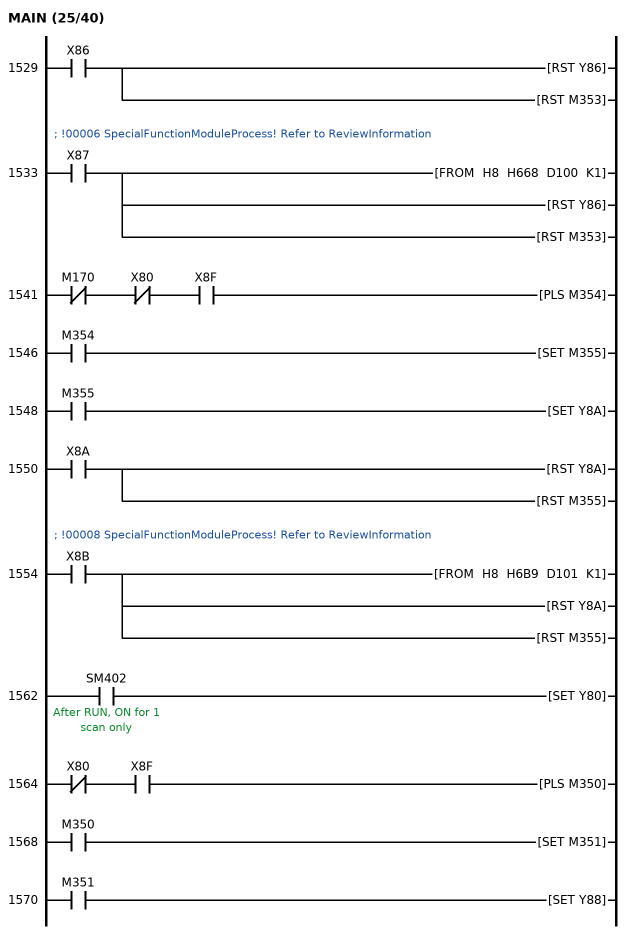
[picture p24: ladder of MAIN, rungs at steps 1529 to 1570]
1529  LD      X86
      RST     Y86
      RST     M353
; !00006 SpecialFunctionModuleProcess! Refer to ReviewInformation
1533  LD      X87
      FROM    H8 H668 D100 K1
      RST     Y86
      RST     M353
1541  LDI     M170
      ANI     X80
      AND     X8F
      PLS     M354
1546  LD      M354
      SET     M355
1548  LD      M355
      SET     Y8A
1550  LD      X8A
      RST     Y8A
      RST     M355
; !00008 SpecialFunctionModuleProcess! Refer to ReviewInformation
1554  LD      X8B
      FROM    H8 H6B9 D101 K1
      RST     Y8A
      RST     M355
1562  LD      SM402  ; After RUN, ON for 1 scan only
      SET     Y80
1564  LDI     X80
      AND     X8F
      PLS     M350
1568  LD      M350
      SET     M351
1570  LD      M351
      SET     Y88
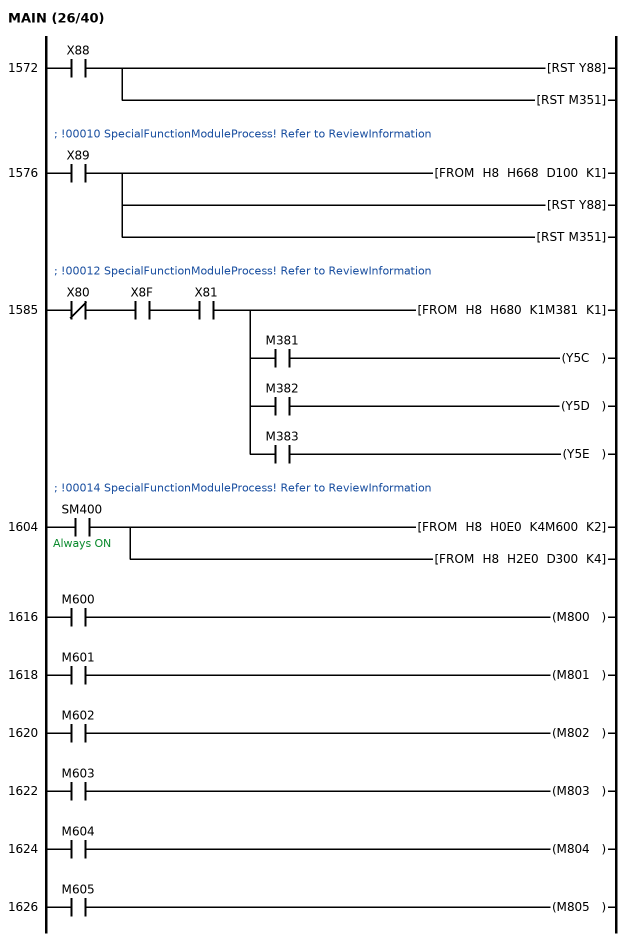
1572  LD      X88
      RST     Y88
      RST     M351
; !00010 SpecialFunctionModuleProcess! Refer to ReviewInformation
1576  LD      X89
      FROM    H8 H668 D100 K1
      RST     Y88
      RST     M351
; !00012 SpecialFunctionModuleProcess! Refer to ReviewInformation
1585  LDI     X80
      AND     X8F
      AND     X81
      FROM    H8 H680 K1M381 K1
      MPS
      AND     M381
      OUT     Y5C
      MRD
      AND     M382
      OUT     Y5D
      MPP
      AND     M383
      OUT     Y5E
; !00014 SpecialFunctionModuleProcess! Refer to ReviewInformation
1604  LD      SM400  ; Always ON
      FROM    H8 H0E0 K4M600 K2
      FROM    H8 H2E0 D300 K4
1616  LD      M600
      OUT     M800
1618  LD      M601
      OUT     M801
1620  LD      M602
      OUT     M802
1622  LD      M603
      OUT     M803
1624  LD      M604
      OUT     M804
1626  LD      M605
      OUT     M805
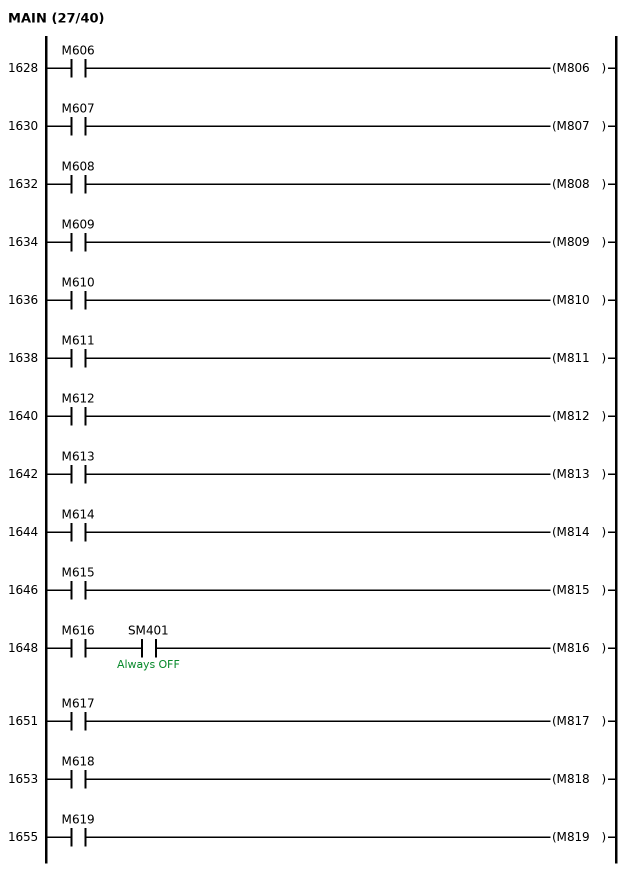
1628  LD      M606
      OUT     M806
1630  LD      M607
      OUT     M807
1632  LD      M608
      OUT     M808
1634  LD      M609
      OUT     M809
1636  LD      M610
      OUT     M810
1638  LD      M611
      OUT     M811
1640  LD      M612
      OUT     M812
1642  LD      M613
      OUT     M813
1644  LD      M614
      OUT     M814
1646  LD      M615
      OUT     M815
1648  LD      M616
      AND     SM401  ; Always OFF
      OUT     M816
1651  LD      M617
      OUT     M817
1653  LD      M618
      OUT     M818
1655  LD      M619
      OUT     M819
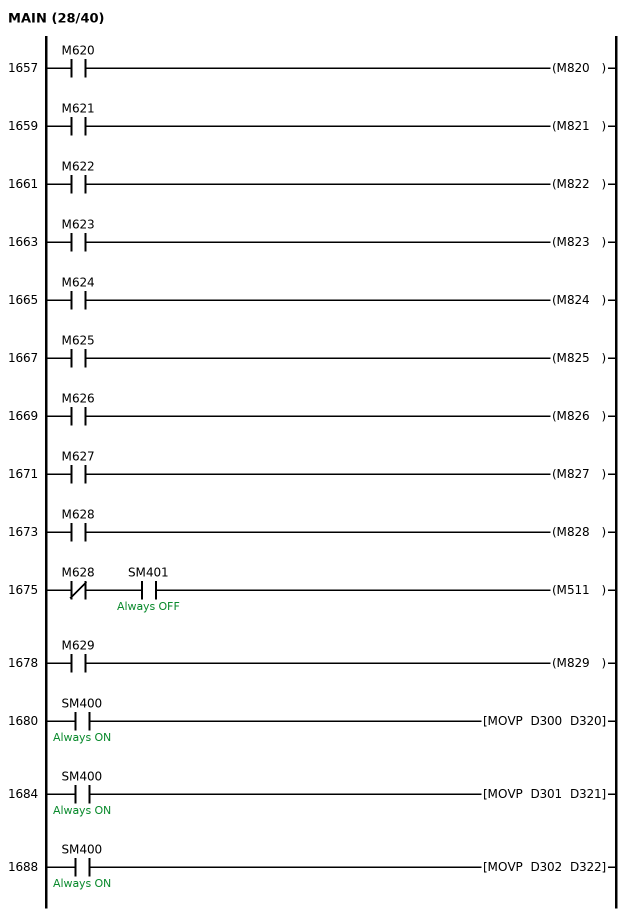
1657  LD      M620
      OUT     M820
1659  LD      M621
      OUT     M821
1661  LD      M622
      OUT     M822
1663  LD      M623
      OUT     M823
1665  LD      M624
      OUT     M824
1667  LD      M625
      OUT     M825
1669  LD      M626
      OUT     M826
1671  LD      M627
      OUT     M827
1673  LD      M628
      OUT     M828
1675  LDI     M628
      AND     SM401  ; Always OFF
      OUT     M511
1678  LD      M629
      OUT     M829
1680  LD      SM400  ; Always ON
      MOVP    D300 D320
1684  LD      SM400  ; Always ON
      MOVP    D301 D321
1688  LD      SM400  ; Always ON
      MOVP    D302 D322
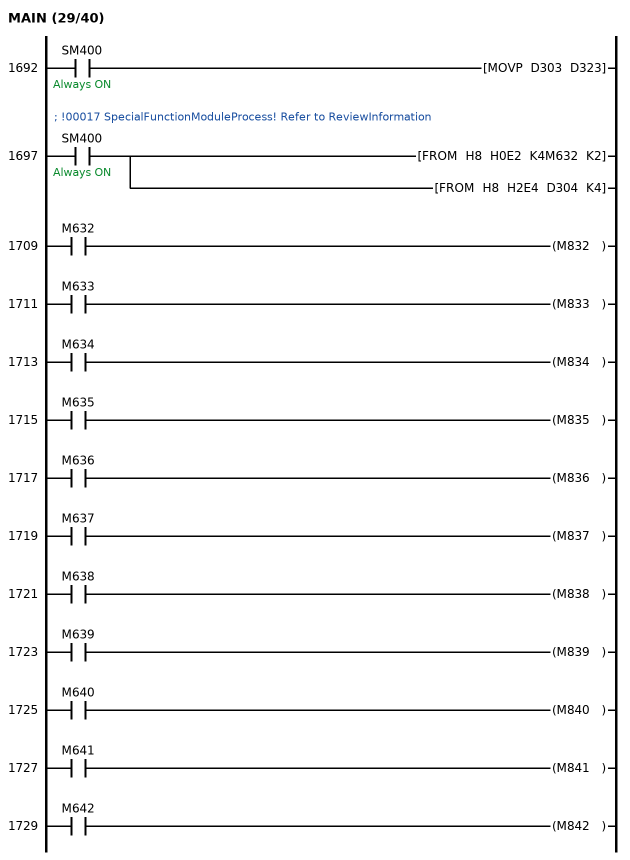
1692  LD      SM400  ; Always ON
      MOVP    D303 D323
; !00017 SpecialFunctionModuleProcess! Refer to ReviewInformation
1697  LD      SM400  ; Always ON
      FROM    H8 H0E2 K4M632 K2
      FROM    H8 H2E4 D304 K4
1709  LD      M632
      OUT     M832
1711  LD      M633
      OUT     M833
1713  LD      M634
      OUT     M834
1715  LD      M635
      OUT     M835
1717  LD      M636
      OUT     M836
1719  LD      M637
      OUT     M837
1721  LD      M638
      OUT     M838
1723  LD      M639
      OUT     M839
1725  LD      M640
      OUT     M840
1727  LD      M641
      OUT     M841
1729  LD      M642
      OUT     M842
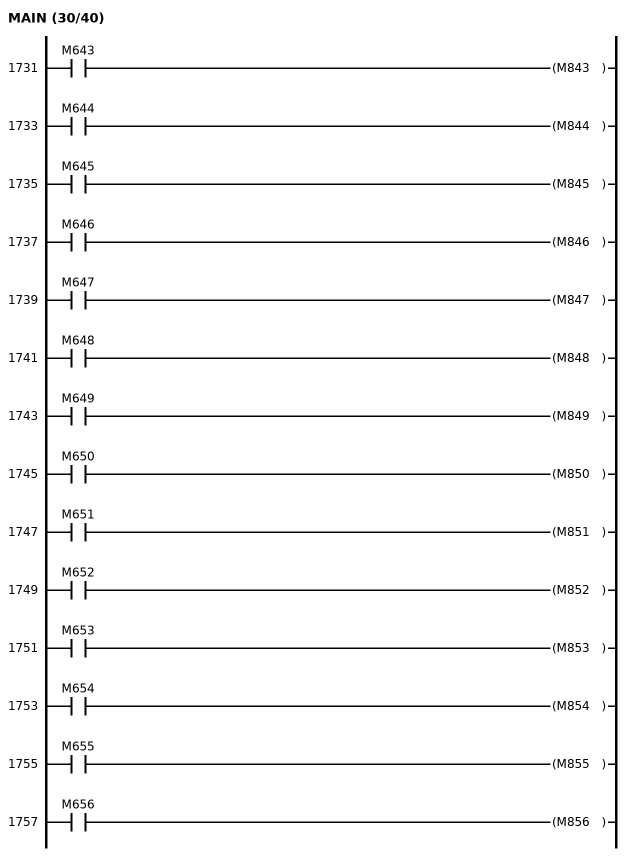
1731  LD      M643
      OUT     M843
1733  LD      M644
      OUT     M844
1735  LD      M645
      OUT     M845
1737  LD      M646
      OUT     M846
1739  LD      M647
      OUT     M847
1741  LD      M648
      OUT     M848
1743  LD      M649
      OUT     M849
1745  LD      M650
      OUT     M850
1747  LD      M651
      OUT     M851
1749  LD      M652
      OUT     M852
1751  LD      M653
      OUT     M853
1753  LD      M654
      OUT     M854
1755  LD      M655
      OUT     M855
1757  LD      M656
      OUT     M856
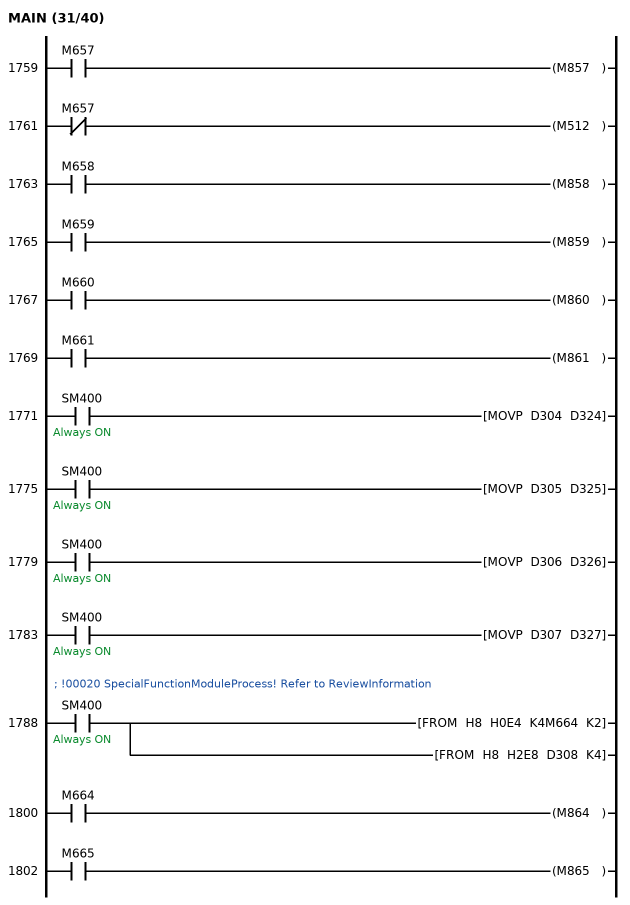
1759  LD      M657
      OUT     M857
1761  LDI     M657
      OUT     M512
1763  LD      M658
      OUT     M858
1765  LD      M659
      OUT     M859
1767  LD      M660
      OUT     M860
1769  LD      M661
      OUT     M861
1771  LD      SM400  ; Always ON
      MOVP    D304 D324
1775  LD      SM400  ; Always ON
      MOVP    D305 D325
1779  LD      SM400  ; Always ON
      MOVP    D306 D326
1783  LD      SM400  ; Always ON
      MOVP    D307 D327
; !00020 SpecialFunctionModuleProcess! Refer to ReviewInformation
1788  LD      SM400  ; Always ON
      FROM    H8 H0E4 K4M664 K2
      FROM    H8 H2E8 D308 K4
1800  LD      M664
      OUT     M864
1802  LD      M665
      OUT     M865
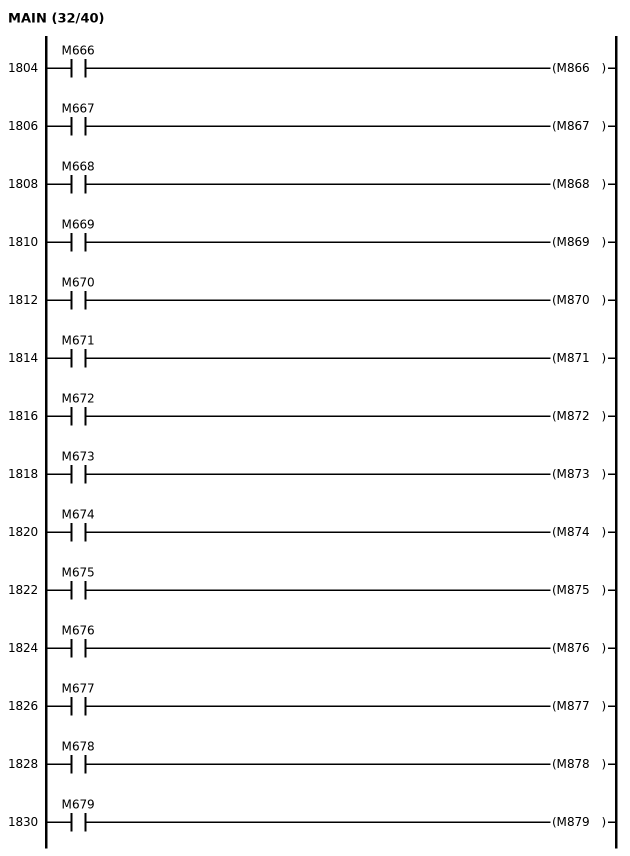
1804  LD      M666
      OUT     M866
1806  LD      M667
      OUT     M867
1808  LD      M668
      OUT     M868
1810  LD      M669
      OUT     M869
1812  LD      M670
      OUT     M870
1814  LD      M671
      OUT     M871
1816  LD      M672
      OUT     M872
1818  LD      M673
      OUT     M873
1820  LD      M674
      OUT     M874
1822  LD      M675
      OUT     M875
1824  LD      M676
      OUT     M876
1826  LD      M677
      OUT     M877
1828  LD      M678
      OUT     M878
1830  LD      M679
      OUT     M879
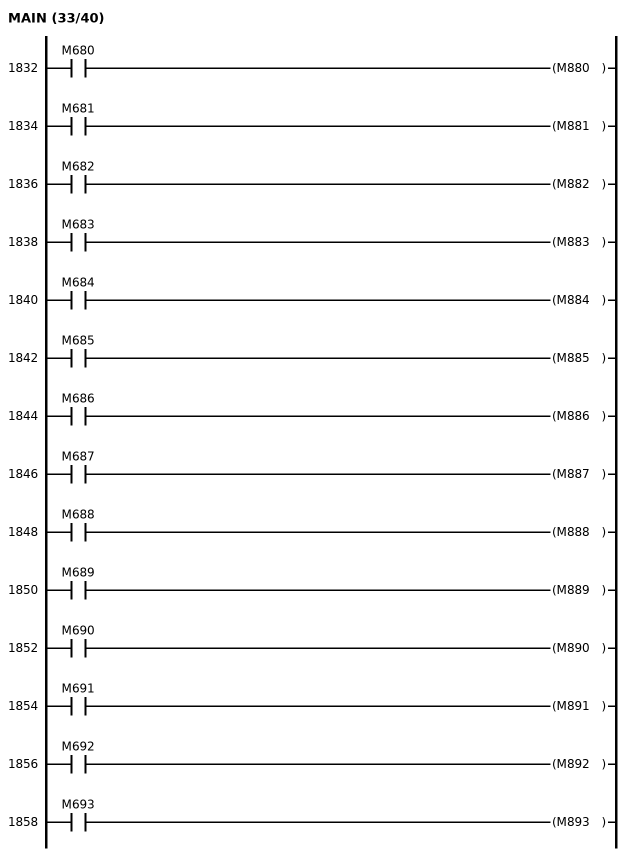
1832  LD      M680
      OUT     M880
1834  LD      M681
      OUT     M881
1836  LD      M682
      OUT     M882
1838  LD      M683
      OUT     M883
1840  LD      M684
      OUT     M884
1842  LD      M685
      OUT     M885
1844  LD      M686
      OUT     M886
1846  LD      M687
      OUT     M887
1848  LD      M688
      OUT     M888
1850  LD      M689
      OUT     M889
1852  LD      M690
      OUT     M890
1854  LD      M691
      OUT     M891
1856  LD      M692
      OUT     M892
1858  LD      M693
      OUT     M893
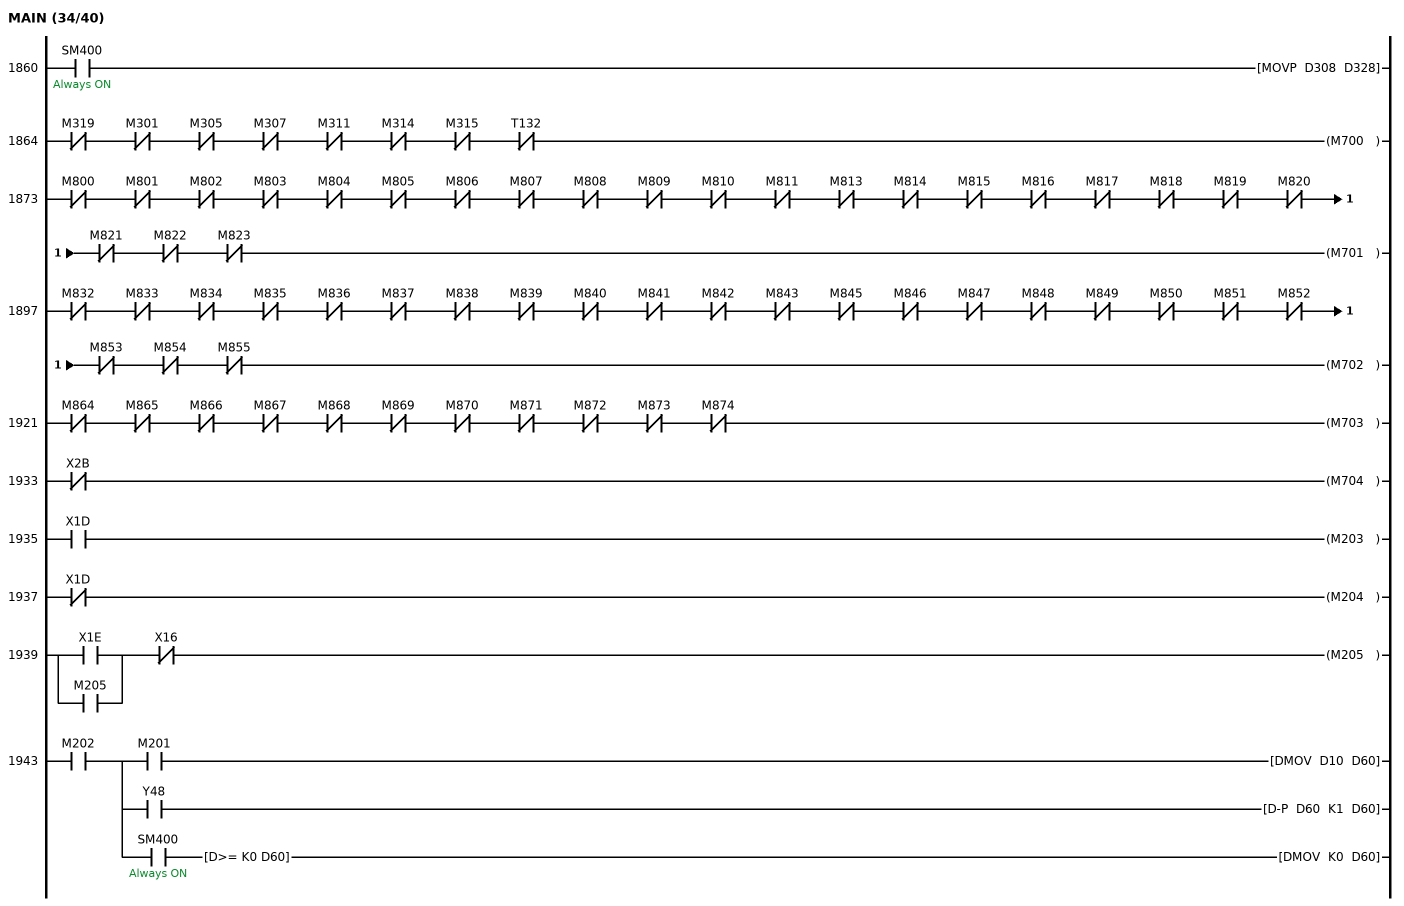
1860  LD      SM400  ; Always ON
      MOVP    D308 D328
1864  LDI     M319
      ANI     M301
      ANI     M305
      ANI     M307
      ANI     M311
      ANI     M314
      ANI     M315
      ANI     T132
      OUT     M700
1873  LDI     M800
      ANI     M801
      ANI     M802
      ANI     M803
      ANI     M804
      ANI     M805
      ANI     M806
      ANI     M807
      ANI     M808
      ANI     M809
      ANI     M810
      ANI     M811
      ANI     M813
      ANI     M814
      ANI     M815
      ANI     M816
      ANI     M817
      ANI     M818
      ANI     M819
      ANI     M820
      ANI     M821
      ANI     M822
      ANI     M823
      OUT     M701
1897  LDI     M832
      ANI     M833
      ANI     M834
      ANI     M835
      ANI     M836
      ANI     M837
      ANI     M838
      ANI     M839
      ANI     M840
      ANI     M841
      ANI     M842
      ANI     M843
      ANI     M845
      ANI     M846
      ANI     M847
      ANI     M848
      ANI     M849
      ANI     M850
      ANI     M851
      ANI     M852
      ANI     M853
      ANI     M854
      ANI     M855
      OUT     M702
1921  LDI     M864
      ANI     M865
      ANI     M866
      ANI     M867
      ANI     M868
      ANI     M869
      ANI     M870
      ANI     M871
      ANI     M872
      ANI     M873
      ANI     M874
      OUT     M703
1933  LDI     X2B
      OUT     M704
1935  LD      X1D
      OUT     M203
1937  LDI     X1D
      OUT     M204
1939  LD      X1E
      OR      M205
      ANI     X16
      OUT     M205
1943  LD      M202
      MPS
      AND     M201
      DMOV    D10 D60
      MRD
      AND     Y48
      D-P     D60 K1 D60
      MPP
      AND     SM400  ; Always ON
      ANDD>=  K0 D60
      DMOV    K0 D60
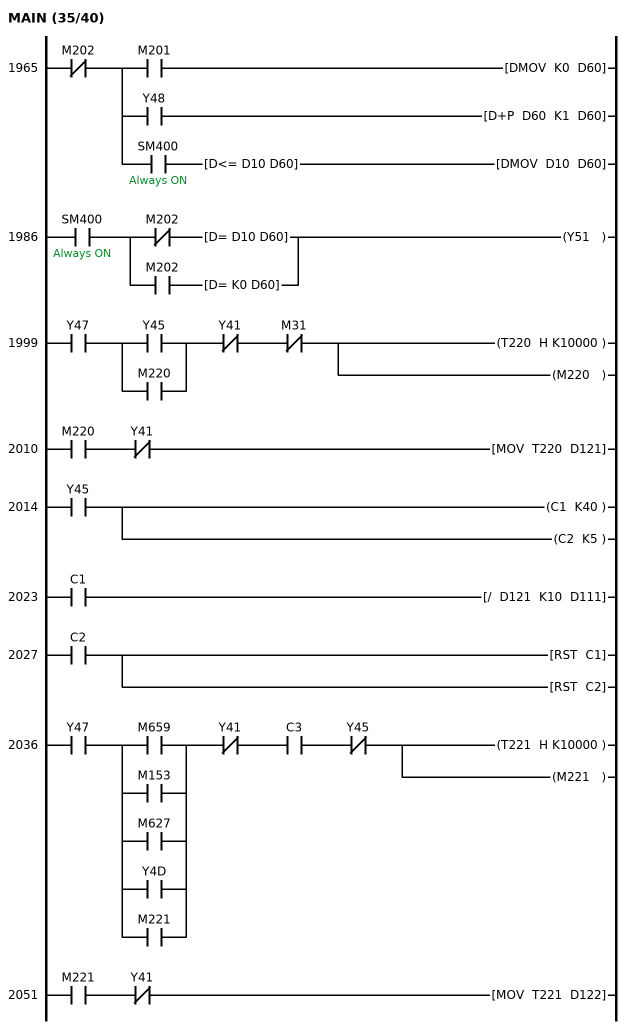
1965  LDI     M202
      MPS
      AND     M201
      DMOV    K0 D60
      MRD
      AND     Y48
      D+P     D60 K1 D60
      MPP
      AND     SM400  ; Always ON
      ANDD<=  D10 D60
      DMOV    D10 D60
1986  LD      SM400  ; Always ON
      LDI     M202
      ANDD=   D10 D60
      LD      M202
      ANDD=   K0 D60
      ORB
      ANB
      OUT     Y51
1999  LD      Y47
      LD      Y45
      OR      M220
      ANB
      ANI     Y41
      ANI     M31
      OUTH    T220 K10000
      OUT     M220
2010  LD      M220
      ANI     Y41
      MOV     T220 D121
2014  LD      Y45
      OUT     C1 K40
      OUT     C2 K5
2023  LD      C1
      /       D121 K10 D111
2027  LD      C2
      RST     C1
      RST     C2
2036  LD      Y47
      LD      M659
      OR      M153
      OR      M627
      OR      Y4D
      OR      M221
      ANB
      ANI     Y41
      AND     C3
      ANI     Y45
      OUTH    T221 K10000
      OUT     M221
2051  LD      M221
      ANI     Y41
      MOV     T221 D122
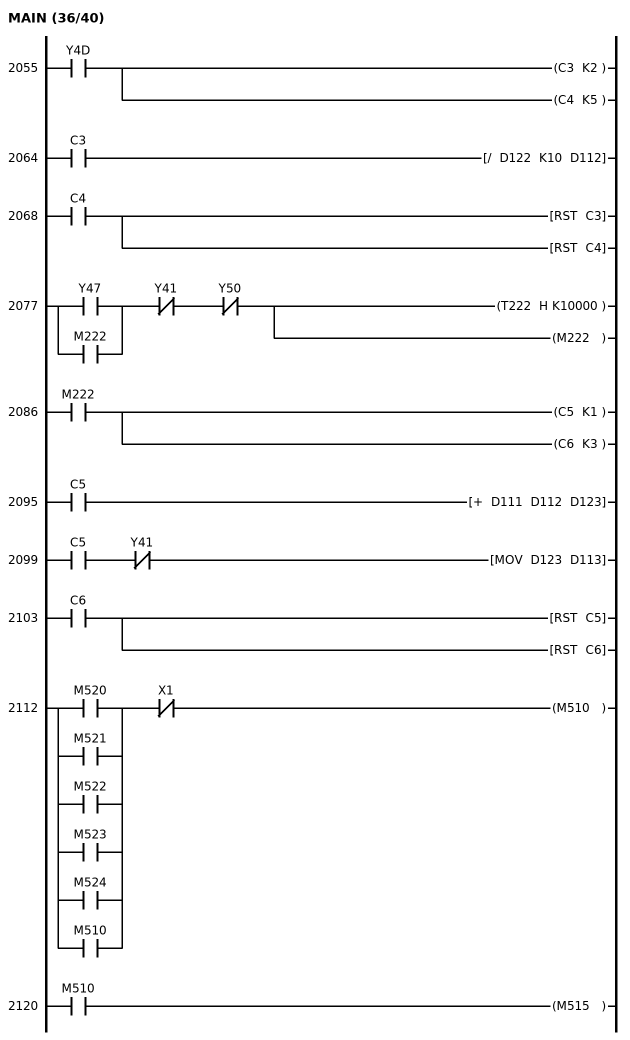
2055  LD      Y4D
      OUT     C3 K2
      OUT     C4 K5
2064  LD      C3
      /       D122 K10 D112
2068  LD      C4
      RST     C3
      RST     C4
2077  LD      Y47
      OR      M222
      ANI     Y41
      ANI     Y50
      OUTH    T222 K10000
      OUT     M222
2086  LD      M222
      OUT     C5 K1
      OUT     C6 K3
2095  LD      C5
      +       D111 D112 D123
2099  LD      C5
      ANI     Y41
      MOV     D123 D113
2103  LD      C6
      RST     C5
      RST     C6
2112  LD      M520
      OR      M521
      OR      M522
      OR      M523
      OR      M524
      OR      M510
      ANI     X1
      OUT     M510
2120  LD      M510
      OUT     M515
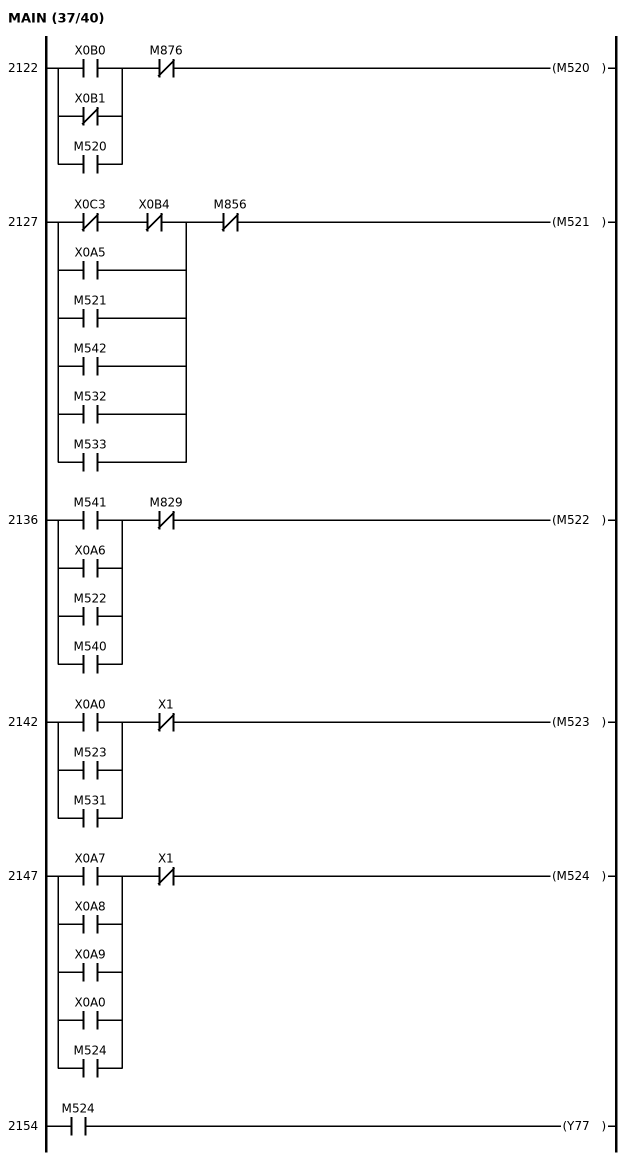
2122  LD      X0B0
      ORI     X0B1
      OR      M520
      ANI     M876
      OUT     M520
2127  LDI     X0C3
      ANI     X0B4
      OR      X0A5
      OR      M521
      OR      M542
      OR      M532
      OR      M533
      ANI     M856
      OUT     M521
2136  LD      M541
      OR      X0A6
      OR      M522
      OR      M540
      ANI     M829
      OUT     M522
2142  LD      X0A0
      OR      M523
      OR      M531
      ANI     X1
      OUT     M523
2147  LD      X0A7
      OR      X0A8
      OR      X0A9
      OR      X0A0
      OR      M524
      ANI     X1
      OUT     M524
2154  LD      M524
      OUT     Y77
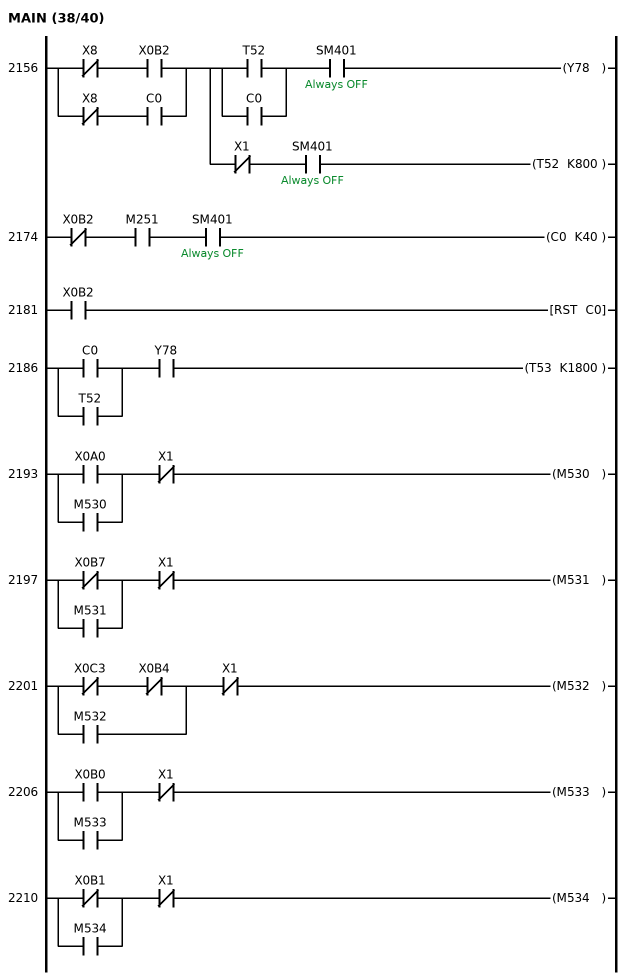
2156  LDI     X8
      AND     X0B2
      LDI     X8
      AND     C0
      ORB
      MPS
      LD      T52
      OR      C0
      ANB
      AND     SM401  ; Always OFF
      OUT     Y78
      MPP
      ANI     X1
      AND     SM401  ; Always OFF
      OUT     T52 K800
2174  LDI     X0B2
      AND     M251
      AND     SM401  ; Always OFF
      OUT     C0 K40
2181  LD      X0B2
      RST     C0
2186  LD      C0
      OR      T52
      AND     Y78
      OUT     T53 K1800
2193  LD      X0A0
      OR      M530
      ANI     X1
      OUT     M530
2197  LDI     X0B7
      OR      M531
      ANI     X1
      OUT     M531
2201  LDI     X0C3
      ANI     X0B4
      OR      M532
      ANI     X1
      OUT     M532
2206  LD      X0B0
      OR      M533
      ANI     X1
      OUT     M533
2210  LDI     X0B1
      OR      M534
      ANI     X1
      OUT     M534
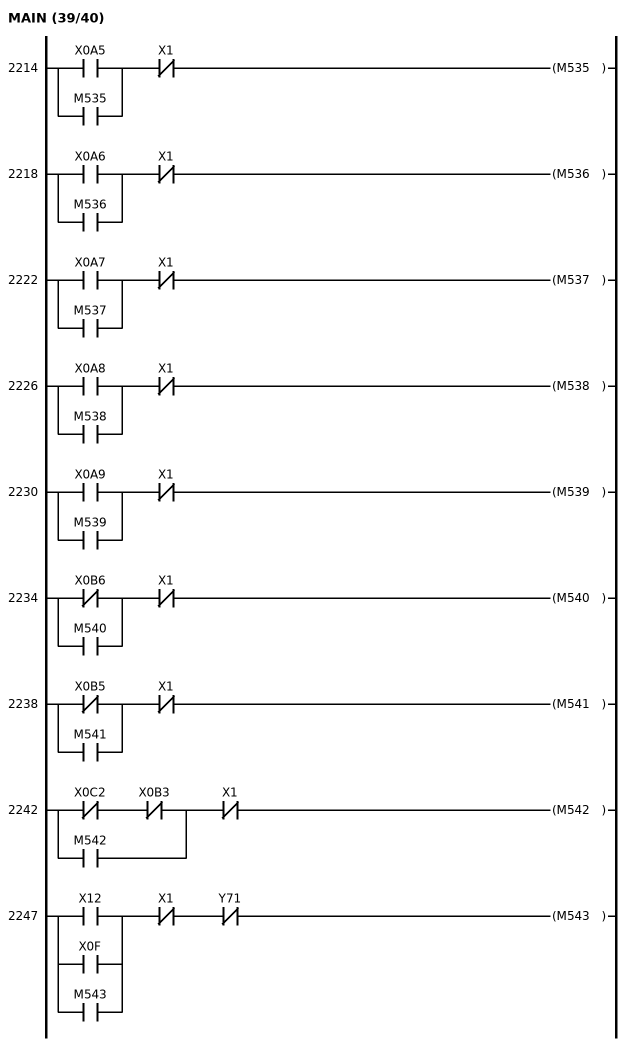
2214  LD      X0A5
      OR      M535
      ANI     X1
      OUT     M535
2218  LD      X0A6
      OR      M536
      ANI     X1
      OUT     M536
2222  LD      X0A7
      OR      M537
      ANI     X1
      OUT     M537
2226  LD      X0A8
      OR      M538
      ANI     X1
      OUT     M538
2230  LD      X0A9
      OR      M539
      ANI     X1
      OUT     M539
2234  LDI     X0B6
      OR      M540
      ANI     X1
      OUT     M540
2238  LDI     X0B5
      OR      M541
      ANI     X1
      OUT     M541
2242  LDI     X0C2
      ANI     X0B3
      OR      M542
      ANI     X1
      OUT     M542
2247  LD      X12
      OR      X0F
      OR      M543
      ANI     X1
      ANI     Y71
      OUT     M543
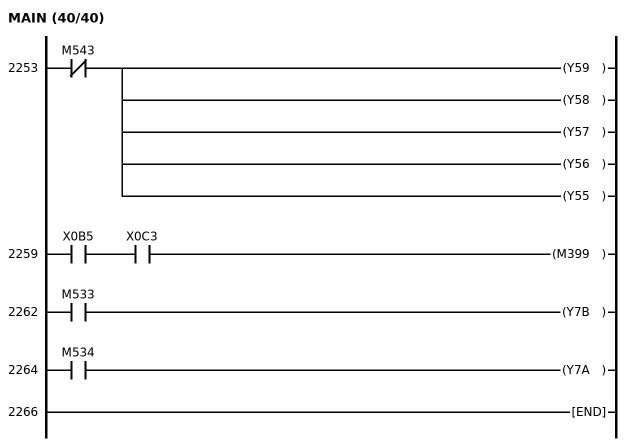
2253  LDI     M543
      OUT     Y59
      OUT     Y58
      OUT     Y57
      OUT     Y56
      OUT     Y55
2259  LD      X0B5
      AND     X0C3
      OUT     M399
2262  LD      M533
      OUT     Y7B
2264  LD      M534
      OUT     Y7A
2266  END
END_PROGRAM
